{region '#Template'}
	{attribute 'Version' := '1.0.0.0'}
	{attribute 'Tags' := '"LCID": "1031", "Text": "DUT, Operation mode, Universal, 3Point"'}
	{attribute 'Tags' := '"LCID": "1033", "Text": "DUT, Operation mode, Universal, 3Point"'}
	{attribute 'Description' := '"LCID": "1031", "Text": "Betriebsart 3 Punkt"'}
	{attribute 'Description' := '"LCID": "1033", "Text": "Operating mode 3 point"'}
{endregion}

{attribute 'qualified_only'}
TYPE E_BA_3Point :
(
	eOff			:= 1,
	eOpen			:= 2,
	eClose			:= 3
	
) UDINT;
END_TYPE

(* stored: Version 1.1.0.1, ProductVersion 3.1.4024.9
   DUT E_BA_3Point: Id {30f61e74-19c1-4e0b-8543-228da9efa94d} *)
